TYPE
    ST_CSV_Step : STRUCT
        seqName     : E_CommandName;
        seqID       : UDINT;
        DetailCount : UDINT;
        Details     : ARRAY[1..MAX_DETAIL_COUNT] OF ST_CSV_Detail;
    END_STRUCT
END_TYPE

(* stored: Version 1.1.0.1
   DUT ST_CSV_Step: Id {afa21cdd-b518-4285-8570-7ac75e658d65} *)
